// :Description: Global parameters for the sample project.
VAR_GLOBAL CONSTANT
    nMaxRetries    : INT := 3;
    fTimeout       : LREAL := 5.0;    (* seconds *)
    sProjectName   : STRING := 'TcKit Sample';
END_VAR

(* stored: Version 1.1.0.1, ProductVersion 3.1.4026.0
   GVL GVL_Params: Id {12345678-0000-0000-0000-000000000010} *)
